// TIA Portal V16 export
// export: Created 2020-12-17T10:32:03.2916545Z, ExportSetting WithDefaults, DisplayName Totally Integrated Automation Portal, DisplayVersion V16 Update 2, DisplayName TIA Portal Version Control Interface, DisplayVersion V16 Update 2, DisplayName TIA Portal Openness, DisplayVersion V16 Update 2, DisplayName STEP 7 Professional, DisplayVersion V16 Update 2, DisplayName STEP 7 Safety, DisplayVersion V16, DisplayName WinCC Advanced / Unified PC, DisplayVersion V16 Update 2
FUNCTION_BLOCK "XBlock_1"   // FB1, FBD
{ S7_Optimized_Access := 'TRUE' }
VERSION : 0.1
// stored: AutoNumber true, IsIECCheckEnabled false, IsRetainMemResEnabled false, MemoryReserve 100, SetENOAutomatically false, UDAEnableTagReadback false
   VAR_INPUT
      iEnable : Bool;
      iStart : Int;
   END_VAR
   VAR_OUTPUT
      qCounter : Int;
   END_VAR
   VAR
      sCounter : Int;
   END_VAR
   VAR CONSTANT
      C_ADD : Int := 1;
   END_VAR
BEGIN

REGION Network 1
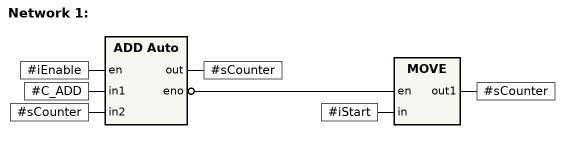
   IF #iEnable THEN #sCounter := #C_ADD + #sCounter; END_IF;
   IF NOT #iEnable THEN #sCounter := #iStart; END_IF;
END_REGION
END_FUNCTION_BLOCK
